TYPE ST_PoseLREAL :
STRUCT
	R_Mat : TcVnMatrix3x3_LREAL;
    T_Mat : TcVnVector3_LREAL;
	X_Mat : TcVnMatrix;
END_STRUCT
END_TYPE

(* stored: Version 1.1.0.1
   DUT ST_PoseLREAL: Id {54128b47-2bd8-4eb0-8d8a-a22074e8cdeb} *)
